# EPICS substitutions: TagApp/Db/readwrite.substitutions
file "readwrite.template" {

# PV name is $(Sys)$(Dev)$(Attr)

# UUID describes the sensor to be read; must be read/write type
#	EPICS doesn't like mixing numbers and letters for some reason, so hex is converted to decimal.
#	eg. 180F -> 18015
# http://processors.wiki.ti.com/index.php/CC2650_SensorTag_User's_Guide

# "Next" points to forward link PV

pattern { Sys, 	Dev  		  ,	Attr 		 , UUID,	Next}
#{ "XF:10IDB",	"{TAG:001}",	"Temperature", "1", 	""}

}
